RoboDK station: Pick Plaque.rdk

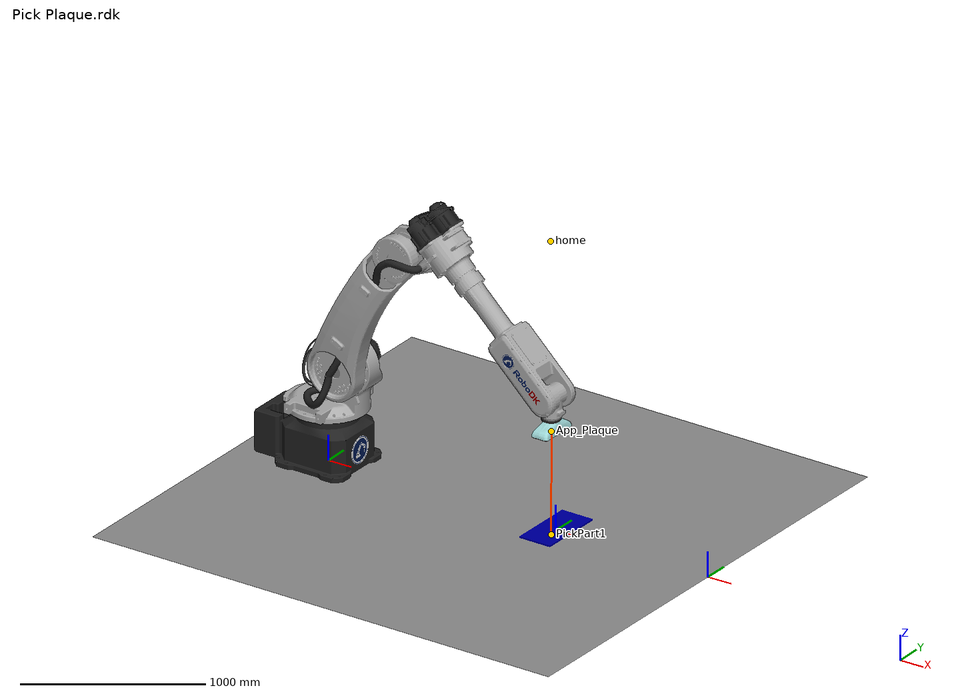
[picture v0: the station drawn from its stored meshes, robots at their saved joint values, targets as dots, program paths as lines]
Station Pick Plaque (saved by RoboDK 6.0.5). Poses are relative to the parent item; angles as X-Y-Z fixed-axis rotations.
  - frame RoboDK RDK-2200 Base at (-1000, 0, 0) mm
    - robot RoboDK RDK-2200: 6 axes
        modified DH rows (alpha deg, a mm, theta deg, d mm): 0, 0, 0, 630; -90, 150, -90, 0; 0, 880, 0, 0; -90, 210, 0, 1105; 90, 0, 0, 0; -90, 0, 180, 140
        joint limits [-180, -90, -110, -180, -125, -360] to [180, 140, 85, 180, 125, 360]; home [0, 0, 0, 0, 0, 0]; saved at [-1.098, 26.529, 16.869, -0.138, 46.586, -271.003]
      - tool Vaccum, TCP at (0, 0, 69.67) mm, size 247.5 x 110 x 75.9 mm
  - frame WORLD at (1500, 0, 0) mm
    - object Floor at (-1500, 0, 0) mm, size 3000 x 3000 x 0 mm, geometry from Floor.sld
    - target home (Cartesian target) at (-1035.33, 0, 1720) mm, rotated rx 0 ry 90 rz 0 deg; joints [0, 0, 0, 0, 0, 0] of RoboDK RDK-2200
  - frame Part1 at (500, 0, 0) mm
    - target App_Plaque (Cartesian target) at (-10, -28.92, 601.04) mm, rotated rx -180 ry 0.1 rz 90 deg; joints [0.289, 25.25, 16.459, -0.134, 48.291, -269.622] of RoboDK RDK-2200
    - target PickPart1 (Cartesian target) at (-10, -30, -20) mm, rotated rx -180 ry 0.1 rz 90 deg; joints [0.247, 53.339, 13.106, -0.25, 23.556, -269.523] of RoboDK RDK-2200
  - program PickPart1 (5 instructions, listed below)
  - program ReplacerObjets (1 instructions, listed below)
  - program PlacePart1 (6 instructions, listed below)
  - object Plaque at (400, 200, 5) mm, rotated rx 0 ry 0 rz -90 deg, size 400 x 200 x 10 mm, geometry from Plaque.sld

--- program PickPart1 (robot RoboDK RDK-2200) ---
  Définir Ref.: Part1
  MoveJ (App_Plaque)
  MoveL (PickPart1)
  Attacher à Vaccum
  MoveL (App_Plaque)

--- program ReplacerObjets (robot RoboDK RDK-2200) ---
  Déplacer Plaque

--- program PlacePart1 (robot RoboDK RDK-2200) ---
  Définir Ref.: Part1
  Choisir Outil: Vaccum
  MoveJ (App_Plaque)
  MoveL (PickPart1)
  Détachez de Vaccum
  MoveL (App_Plaque)
